PROGRAM FeedMotor2Manualcontrol
VAR
END_VAR

// Written 10.08.2023 by Daniel Kelly

// Program provides manual control of the removal motor M2 via its switch

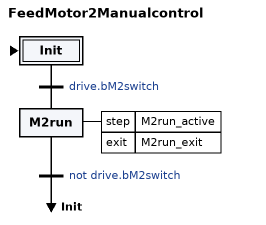
INITIAL_STEP Init:
END_STEP
TRANSITION FROM Init TO M2run
    := drive.bM2switch;
END_TRANSITION
STEP M2run:
    M2run_active(N);  // step action
    M2run_exit(P0);  // exit action
END_STEP
TRANSITION FROM M2run TO Init
    := not drive.bM2switch;
END_TRANSITION

ACTION M2run_active:
drive.bRemovalMotor := TRUE;
END_ACTION

ACTION M2run_exit:
drive.bRemovalMotor := FALSE;
END_ACTION

ACTION manualCTRL2_active:
drive.bRemovalMotor := TRUE; 
drive.bM2active := TRUE;
END_ACTION

ACTION manualCTRL2_entry:
//drive.bRemovalMotor := TRUE; 
//drive.bM2active := TRUE;
END_ACTION

ACTION manualCTRL2_exit:
drive.bRemovalMotor := FALSE; 
drive.bM2active := FALSE;
END_ACTION

END_PROGRAM

(* stored: Version 1.1.0.1, ProductVersion 3.1.4024.12
   POU FeedMotor2Manualcontrol: Id {4830c5b8-1733-4acc-96dd-e5817fad03dc}, SpecialFunc None
   Action M2run_active: Id {f26f3304-40b8-4f7f-b9de-eb12dda2024e}
   Action M2run_exit: Id {4c552573-7e4e-4bfa-8d03-6f5b444b9e9c}
   Action manualCTRL2_active: Id {f196b1cf-0fe7-4087-8eb5-f98b1da133a6}
   Action manualCTRL2_entry: Id {b383cb7a-e1c2-4ba0-82a0-97d2ec4e8639}
   Action manualCTRL2_exit: Id {48fffafa-213d-48d2-bcfa-0bf9cfd9b911} *)
